(* CODESYS project CtaAppIO_2.0.0.0.library
   Description: Io Applikation Library der CTA
   Version: 2.0.0.0
   Title: CtaAppIO
   Author: SIS
   DocFormat: reStructuredText
   LanguageModelAttribute: qualified-access-only
   Placeholder: CtaAppIO
   DefaultNamespace: CtaAppIO
   CompiledLibraryCompatibilityVersion: CODESYS V3.5 SP16 Patch 3
   Company: CTA

Project tree, tasks and I/O mapping:
  libraries: Standard, 3.5.18.0 (System); CtaVisSymbols, 2.0.0.0 (CTA); VisuSymbols, 4.5.0.0 (System); CtaSysIO, 2.0.0.0 (CTA)
  40 Visualizations/
  30 Program Organization Units/
    AI/
      function fcAI [ST]
      function fcAI_INI [ST]
    DI/
      function fcDI [ST]
      function fcDI_INI [ST]
    AO/
      function fcAO [ST]
      function fcAO_INI [ST]
    DO/
      function fcDO [ST]
      function fcDO_INI [ST]
    IO/
      function fcIO [ST]
    SLOT/
      function fcCheckSlot [ST]
  00000000-0000-0000-0000-000000000000|D:\CoDeSys\LibrariesV3\trunk\Intern\CAA\CAA Template\3.4.0.0 draft\Placeholder.xml
  00000000-0000-0000-0000-000000000000|D:\CoDeSys\LibrariesV3\trunk\Intern\CAA\CAA Template\3.2.0.3 draft\Prefix.pdf
  00000000-0000-0000-0000-000000000000|D:\CoDeSys\LibrariesV3\trunk\Intern\CAA\CAA Template\3.5.2.0 draft\Placeholder.xml
  20 Structs/
  50 Images/
  10 Documenation/
    global variables VersionHistory
    global variables readMe
  21 Interface/
  11 Library Parameter/
  12 Konstanten/
  60 Textlisten/
  13 Globale Variablen/
  text list GlobalTextList
  5ce3da45-db07-42e7-a21c-a00fff4ed8f6|Image\Sortet\0750_432.bmp
  5ce3da45-db07-42e7-a21c-a00fff4ed8f6|Image\Sortet\0750_455.bmp
  5ce3da45-db07-42e7-a21c-a00fff4ed8f6|Image\Sortet\0750_466.bmp
  5ce3da45-db07-42e7-a21c-a00fff4ed8f6|Image\Sortet\0750_597.bmp
  5ce3da45-db07-42e7-a21c-a00fff4ed8f6|Image\Sortet\0750_1405.bmp
  5ce3da45-db07-42e7-a21c-a00fff4ed8f6|Image\Sortet\0750_8212.bmp
  5ce3da45-db07-42e7-a21c-a00fff4ed8f6|C:\Users\sis\Desktop\WagoVisu\Image\Sortet\0750_BLANK.bmp
*)

// 10 Documenation/VersionHistory
(* 

.. image:: ../../Images/CTA_Logo.jpg
   :align: right
   :width: 15% 

**Vorlage**   


============ =========== =========== ============================================
**Date**     **Version** **Author**  **Change**
------------ ----------- ----------- --------------------------------------------
04.03.2021   0.0.0.0     SIS         Vorlage erstellt

============ =========== =========== ============================================


*)
VAR_GLOBAL
    stInfo : STRING:= '0.0.0.0, Vorlage, CTA';
END_VAR

// 10 Documenation/readMe
(*

**ReadMe**
 
|	 **Empfehlung**
|
|	 Bibliothek CtaAppIO zur Verlinkung und Beschaltung von Ein- und Ausgängen
|	 Anwendung der Bibliothek wie Verlinkung und Beschaltung erfolgt wie im Code- Beispiel dargestellt.
|  
| *Beispiel* 

+-----------------------+---------------------------------------------------------------------------------------------------------------------------------------------------------------------------------------------------------------------------------------------------------------------------------------------------------------------------------------------------------------------------------------------------------------------------------------+
| Beschreibung          |  Code                                                                                                                                                                                                                                                                                                                                                                                                                                 |
+=======================+=======================================================================================================================================================================================================================================================================================================================================================================================================================================+
| Initialisierung		| .. code-block:: codesys                                                                                                                                                                                                                                                                                                                                                                                                               |
|                       |                                                                                                                                                                                                                                                                                                                                                                                                                                       |
|                       |	// Analoge Eingänge																																																																																																					|
|                       |	CtaAppIO.fcAI_INI(	_usiDeviceNr		:= 	1,       																																																																																												|
|                       |						_usiSlotNr			:=	2,         																																																																																												|
|                       |						_usiIoNr			:= 	3,          																																																																																											|
|                       |						xSimulationLock		:= 	FALSE,																																																																																													|
|                       |						rMin				:=	 30.0,          																																																																																										|
|                       |						rMax				:=  100.0,         																																																																																											|
|                       |						rMinPhysical		:=    0.0,   																																																																																												|
|                       |						rPhysicalAlarm		:=    0.0, 																																																																																													|
|                       |						rCorrectionValue	:=    0.0,																																																																																													|
|						|                                                                   																																																																																									|
|						|	// Analoge Ausgängen																																																																																																				|
|                       |	CtaAppIO.fcAO_INI(	_usiDeviceNr		:= 	1,																																																																																														|
|                       |						_usiSlotNr			:=	2,                																																																																																										|
|                       |						_usiIoNr			:= 	3,                 																																																																																										|
|                       |						xSimulationLock		:= 	FALSE,       																																																																																											|
|                       |						rMin				:=	 30.0,                 																																																																																									|
|                       |						rMax				:=  100.0,                																																																																																									|
|                       |						rMinPhysical		:=   0.0);         																																																																																											|
|                       |																																																																																																										|
|						|	// Digitale Eingänge																																																																																																				|
|                       |	CtaAppIO.fcDI_INI(	_usiDeviceNr		:= 	1,																																																																																														|
|                       |						_usiSlotNr			:=	2,                																																																																																										|
|                       |						_usiIoNr			:= 	3,                 																																																																																										|
|                       |						xSimulationLock		:= 	FALSE,       																																																																																											|
|                       |						xInvert				:=  FALSE);            																																																																																										|
|						|																																																																																																										|
|						|	// Digitale Ausgänge 																																																																																																				|
|                       |	CtaAppIO.fcDO_INI(	_usiDeviceNr		:= 	1,																																																																																														|
|                       |						_usiSlotNr			:=	2,                																																																																																										|
|                       |						_usiIoNr			:= 	3,                 																																																																																										|
|                       |						xSimulationLock		:= 	FALSE,       																																																																																											|
|                       |						xInvert				:=  FALSE);            																																																																																										|
|                       |																																																																																																										|
+-----------------------+---------------------------------------------------------------------------------------------------------------------------------------------------------------------------------------------------------------------------------------------------------------------------------------------------------------------------------------------------------------------------------------------------------------------------------------+
|Ausführung und Linking	| .. code-block:: codesys                                                                                                                                                                                                                                                                                                                                                                                                               |
|                       |  																																																																																																										|
|						|	//Interface zuweisung (Unabhängig von Modultyp)                                                                       																																																																												|
|						|                                                                                                                         																																																																												|
|						| 		F100.B011.metSetITF(CtaAppIO.fcIO(DeviceNr,SlotNr,IoNr));                                                     																																																																													|
|						|																																																																																																										|
|			 			|	// Direkte Wertzuweisungen (Modul abhängig)                                                                           																																																																												|
|						|                                                                                                                         																																																																												|
|						|		// Analoge Eingänge                                                                                               																																																																												|
|						|                                                                                                                         																																																																												|
|						|			CtaAppIO.fcAI(DeviceNr,SlotNr,IoNr,rAI_Value => POU.Variable);	                                              																																																																												|
|						|		                                                                                                                  																																																																												|
|						|		// Analoge Ausgänge                                                                                               																																																																												|
|						|                                                                                                                         																																																																												|
|						|			CtaAppIO.fcAO(DeviceNr,SlotNr,IoNr,POU.Variable);                                                             																																																																												|
|						|                                                                                                                         																																																																												|
|						|		// Digitale Eingänge                                                                                              																																																																												|
|						|                                                                                                                         																																																																												|
|						|			CtaAppIO.fcDI(DeviceNr,SlotNr,IoNr,xDI_Value => POU.Variable);                                                																																																																												|
|                       |                                                                                                                         																																																																												|
|						|		// Digitale Ausgänge                                                                                              																																																																												|
|						|                                                                                                                         																																																																												|
|						|	     	CtaAppIO.fcDO(DeviceNr,SlotNr,IoNr,POU.Variable);                                                             																																																																												|
|			 			|	                                                                                                                      																																																																												|
+-----------------------+---------------------------------------------------------------------------------------------------------------------------------------------------------------------------------------------------------------------------------------------------------------------------------------------------------------------------------------------------------------------------------------------------------------------------------------+
*)                                                                                                                                                                                                                                                                                                                                                                                                                                                               
VAR_GLOBAL
	xReadMeDone              :   BOOL; 
END_VAR

// 30 Program Organization Units/DI/fcDI
FUNCTION fcDI : BOOL
VAR_INPUT
	_usiDeviceNr		:	USINT;
	_usiSlotNr			: 	USINT;
	_usiIoNr			: 	USINT;
END_VAR
VAR_OUTPUT
	xDI_Value			:	BOOL;
END_VAR
VAR
	ITF_IO		:	CtaSysIO.ITF_IO;
	ITF_DI		:	CtaSysIO.ITF_DI;
END_VAR

ITF_IO := CtaSysIO.GVL_IO.FB_IO_MANAGER.GET_IO(_usiDeviceNr,_usiSlotNr,_usiIoNr);
IF __QUERYINTERFACE(ITF_IO,ITF_DI) THEN
	xDI_Value 	:= ITF_DI.proValue;
	fcDI		:= TRUE;
ELSE
	fcDI		:= FALSE;
END_IF;

END_FUNCTION

// 30 Program Organization Units/AI/fcAI
FUNCTION fcAI : BOOL
VAR_INPUT
	_usiDeviceNr		:	USINT;
	_usiSlotNr			: 	USINT;
	_usiIoNr			: 	USINT;
END_VAR
VAR_OUTPUT
	rAI_Value	:	REAL;
END_VAR
VAR
	ITF_IO		:	CtaSysIO.ITF_IO;
	ITF_AI		:	CtaSysIO.ITF_AI;
END_VAR

ITF_IO := CtaSysIO.GVL_IO.FB_IO_MANAGER.GET_IO(_usiDeviceNr,_usiSlotNr,_usiIoNr);
IF __QUERYINTERFACE(ITF_IO,ITF_AI) THEN
	rAI_Value	:= ITF_AI.proValue;
	fcAI		:= TRUE;
ELSE
	fcAI		:= FALSE;
END_IF;

END_FUNCTION

// 30 Program Organization Units/DO/fcDO
FUNCTION fcDO : BOOL
VAR_INPUT
	_usiDeviceNr		:	USINT;
	_usiSlotNr			: 	USINT;
	_usiIoNr			: 	USINT;
	xDO_Value			:	BOOL;	
END_VAR
VAR
	ITF_IO				:	CtaSysIO.ITF_IO;
	ITF_DO				:	CtaSysIO.ITF_DO;
END_VAR

ITF_IO := CtaSysIO.GVL_IO.FB_IO_MANAGER.GET_IO(_usiDeviceNr,_usiSlotNr,_usiIoNr);
IF __QUERYINTERFACE(ITF_IO,ITF_DO) THEN
	ITF_DO.proValue := xDO_Value;
	fcDO			:= TRUE;
ELSE
	fcDO			:= FALSE;
END_IF;

END_FUNCTION

// 30 Program Organization Units/IO/fcIO
FUNCTION fcIO 	: CtaSysIO.ITF_IO;
VAR_INPUT
	_usiDeviceNr		:	USINT;
	_usiSlotNr			: 	USINT;
	_usiIoNr			: 	USINT;
END_VAR
VAR
END_VAR

fcIO := CtaSysIO.GVL_IO.FB_IO_MANAGER.GET_IO(_usiDeviceNr,_usiSlotNr,_usiIoNr);

END_FUNCTION

// 30 Program Organization Units/AO/fcAO
FUNCTION fcAO : BOOL
VAR_INPUT
	_usiDeviceNr		:	USINT;
	_usiSlotNr			: 	USINT;
	_usiIoNr			: 	USINT;
	rAO_Value	:	REAL;
END_VAR
VAR
	ITF_IO		:	CtaSysIO.ITF_IO;
	ITF_AO		:	CtaSysIO.ITF_AO;
END_VAR

ITF_IO := CtaSysIO.GVL_IO.FB_IO_MANAGER.GET_IO(_usiDeviceNr,_usiSlotNr,_usiIoNr);
IF __QUERYINTERFACE(ITF_IO,ITF_AO) THEN
	ITF_AO.proValue 	:= rAO_Value;
	fcAO				:= TRUE;
ELSE
	fcAO				:= FALSE;
END_IF;

END_FUNCTION

// 30 Program Organization Units/AI/fcAI_INI
FUNCTION fcAI_INI : BOOL
VAR_INPUT
	_usiDeviceNr		:	USINT;
	_usiSlotNr			: 	USINT;
	_usiIoNr			: 	USINT;
	xSimulationLock		:	BOOL;
	rMin				:	REAL;
	rMax				:	REAL;
	rMinPhysical		:	REAL;
	rPhysicalAlarm		:	REAL;
	rCorrectionValue	:	REAL;
	stPhysicalUnit		:	STRING(40);	
END_VAR
VAR
	ITF_DEVICE	:	CtaSysIO.ITF_IO_DEVICE;
	ITF_IO		:	CtaSysIO.ITF_IO;
	ITF_AI		:	CtaSysIO.ITF_AI;
	scAI_Para	:	CtaSysIO.scAI_Para;
END_VAR

ITF_DEVICE := CtaSysIO.GVL_IO.FB_IO_MANAGER.GET_DEVICE(_usiDeviceNr);
IF __QUERYINTERFACE(ITF_DEVICE,ITF_DEVICE) THEN
	IF ITF_DEVICE.GET_STATE_READY_TO_SET_CONFIG THEN
		ITF_IO := CtaSysIO.GVL_IO.FB_IO_MANAGER.GET_IO(_usiDeviceNr,_usiSlotNr,_usiIoNr);
		IF __QUERYINTERFACE(ITF_IO,ITF_AI) THEN
			scAI_Para.xSimulationLock	:= xSimulationLock;
			scAI_Para.rMin				:= rMin;
			scAI_Para.rMax				:= rMax;
			scAI_Para.rMinPhysical		:= rMinPhysical;
			scAI_Para.rPhysicalAlarm	:= rPhysicalAlarm;
			scAI_Para.rCorrectionValue	:= rCorrectionValue;
			scAI_Para.stPhysicalUnit	:= stPhysicalUnit;
			ITF_AI.P_All_Init			:= scAI_Para;
			fcAI_INI					:= TRUE;	
		ELSE
			fcAI_INI					:= FALSE;
		END_IF;
	END_IF;
END_IF;

END_FUNCTION

// 30 Program Organization Units/AO/fcAO_INI
FUNCTION fcAO_INI : BOOL
VAR_INPUT
	_usiDeviceNr		:	USINT;
	_usiSlotNr			: 	USINT;
	_usiIoNr			: 	USINT;
	xSimulationLock		:	BOOL;
	rMin				:	REAL;
	rMax				:	REAL;
	rMinPhysical		:	REAL;
END_VAR
VAR
	ITF_DEVICE	:	CtaSysIO.ITF_IO_DEVICE;
	ITF_IO		:	CtaSysIO.ITF_IO;
	ITF_AO		:	CtaSysIO.ITF_AO;
	scAO_Para	:	CtaSysIO.scAO_Para;
END_VAR

ITF_DEVICE := CtaSysIO.GVL_IO.FB_IO_MANAGER.GET_DEVICE(_usiDeviceNr);
IF __QUERYINTERFACE(ITF_DEVICE,ITF_DEVICE) THEN
	IF ITF_DEVICE.GET_STATE_READY_TO_SET_CONFIG THEN
		ITF_IO := CtaSysIO.GVL_IO.FB_IO_MANAGER.GET_IO(_usiDeviceNr,_usiSlotNr,_usiIoNr);
		IF __QUERYINTERFACE(ITF_IO,ITF_AO) THEN
			scAO_Para.xSimulationLock	:= xSimulationLock;
			scAO_Para.rMin				:= rMin;
			scAO_Para.rMax				:= rMax;
			scAO_Para.rMinPhysical		:= rMinPhysical;
			ITF_AO.P_All_Init			:= scAO_Para;
			fcAO_INI					:= TRUE;	
		ELSE
			fcAO_INI					:= FALSE;
		END_IF;
	END_IF;
END_IF;

END_FUNCTION

// 30 Program Organization Units/DI/fcDI_INI
FUNCTION fcDI_INI : BOOL
VAR_INPUT
	_usiDeviceNr		:	USINT;
	_usiSlotNr			: 	USINT;
	_usiIoNr			: 	USINT;
	xSimulationLock		:	BOOL;
	xInvert				:	BOOL;
END_VAR
VAR
	ITF_DEVICE	:	CtaSysIO.ITF_IO_DEVICE;
	ITF_IO		:	CtaSysIO.ITF_IO;
	ITF_DI		:	CtaSysIO.ITF_DI;
	scDI_Para	:	CtaSysIO.scDI_Para;
END_VAR

ITF_DEVICE := CtaSysIO.GVL_IO.FB_IO_MANAGER.GET_DEVICE(_usiDeviceNr);
IF __QUERYINTERFACE(ITF_DEVICE,ITF_DEVICE) THEN
	IF ITF_DEVICE.GET_STATE_READY_TO_SET_CONFIG THEN
		ITF_IO := CtaSysIO.GVL_IO.FB_IO_MANAGER.GET_IO(_usiDeviceNr,_usiSlotNr,_usiIoNr);
		IF __QUERYINTERFACE(ITF_IO,ITF_DI) THEN
			scDI_Para.xSimulationLock	:= xSimulationLock;
			scDI_Para.xInvert			:= xInvert;
			ITF_DI.P_All_Init			:= scDI_Para;
			fcDI_INI					:= TRUE;	
		ELSE
			fcDI_INI					:= FALSE;
		END_IF;
	END_IF;
END_IF;

END_FUNCTION

// 30 Program Organization Units/DO/fcDO_INI
FUNCTION fcDO_INI : BOOL
VAR_INPUT
	_usiDeviceNr		:	USINT;
	_usiSlotNr			: 	USINT;
	_usiIoNr			: 	USINT;
	xSimulationLock		:	BOOL;
	xInvert				:	BOOL;
END_VAR
VAR
	ITF_DEVICE	:	CtaSysIO.ITF_IO_DEVICE;
	ITF_IO		:	CtaSysIO.ITF_IO;
	ITF_DO		:	CtaSysIO.ITF_DO;
	scDO_Para	:	CtaSysIO.scDO_Para;
END_VAR

ITF_DEVICE := CtaSysIO.GVL_IO.FB_IO_MANAGER.GET_DEVICE(_usiDeviceNr);
IF __QUERYINTERFACE(ITF_DEVICE,ITF_DEVICE) THEN
	IF ITF_DEVICE.GET_STATE_READY_TO_SET_CONFIG THEN
		ITF_IO := CtaSysIO.GVL_IO.FB_IO_MANAGER.GET_IO(_usiDeviceNr,_usiSlotNr,_usiIoNr);
		IF __QUERYINTERFACE(ITF_IO,ITF_DO) THEN
			scDO_Para.xSimulationLock	:= xSimulationLock;
			scDO_Para.xInvert			:= xInvert;
			ITF_DO.P_All_Init			:= scDO_Para;
			fcDO_INI					:= TRUE;	
		ELSE
			fcDO_INI					:= FALSE;
		END_IF;
	END_IF;
END_IF;

END_FUNCTION

// 30 Program Organization Units/SLOT/fcCheckSlot
FUNCTION fcCheckSlot : BOOL
VAR_INPUT
	_usiDeviceNr		:	USINT;
	_usiSlotNr			: 	USINT;
	enCheckIoIn			:	CtaSysIO.enCheckIo;
	usiAnzIoType		:	USINT;
	enSimIoTypeIn		:	CtaSysIO.enIOType := CtaSysIO.enIOType.Unknown;
END_VAR

CtaSysIO.GVL_IO.FB_IO_MANAGER.CHECK_SLOT(_usiDeviceNr,_usiSlotNr,enCheckIoIn,enSimIoTypeIn,usiAnzIoType);

END_FUNCTION
